FUNCTION_BLOCK PUBLIC LtiBasicAxis_FB EXTENDS CoE_BasicAxis_FB  
VAR_INPUT		
	pDigIn: 	POINTER TO DINT;
END_VAR
VAR_IN_OUT	
END_VAR
VAR_OUTPUT	
END_VAR

VAR
	
	
END_VAR



SUPER^(AxisRef:=AxisRef);

METHOD GetErrCanAdr : BOOL
VAR_INPUT
END_VAR


VAR
		
END_VAR
SUPER^.GetCanOpenAdr();		
CoeErrIdIndex	 := 16#2027;
CoeErrIdSubIndex := 0;
END_METHOD

METHOD ReadActualTorque : LREAL
VAR_INPUT
END_VAR
VAR_INST
	
	
	
END_VAR

IF THIS^.TorqueReadEnable THEN			
	tmp_ActualTorque:= io_ActualTorqueReal;		
END_IF

ReadActualTorque:= tmp_ActualTorque;
END_METHOD

METHOD ReadDriveError
VAR_INPUT
END_VAR
VAR_INST 
	ErrIdIndex	: WORD;
END_VAR
DriveError := AxisRef.NcToPlc.StateDWord AND 16#10000000 ;
ErrIdIndex	:= 16#2027; // decimal = 39;
END_METHOD

END_FUNCTION_BLOCK

(* stored: Version 1.1.0.1, ProductVersion 3.1.4024.3
   POU LtiBasicAxis_FB: Id {58c8b0ec-012c-067f-0bc8-f751a305a480}, SpecialFunc None
   Method GetErrCanAdr: Id {498aeda4-df0d-0abc-1512-6585c242e02a}
   Method ReadActualTorque: Id {92742f0d-b1f8-0eb5-1cbc-7a5bc6013b51}
   Method ReadDriveError: Id {86d63129-2d10-09d1-23bb-cc7808e46b63} *)
